{attribute addProperty BoxType "EL6861-0000-0016"}
{attribute addProperty Id "Transmit_requestBIT10.1251Receive_acceptedBIT10.1252Init_requestBIT10.1253Send_continuousBIT10.1254Output_lenUSINT819"}
{attribute addProperty CRC "829288253"}
{attribute addProperty SizeInBites "16"}
{attribute addProperty SizeInBytes "2"}
TYPE Ctrl_316DEF3D :
STRUCT
	{attribute addProperty Name "Transmit_request"}
	Transmit_request : BIT;
	{attribute addProperty Name "Receive_accepted"}
	Receive_accepted : BIT;
	{attribute addProperty Name "Init_request"}
	Init_request : BIT;
	{attribute addProperty Name "Send_continuous"}
	Send_continuous : BIT;
	{attribute 'hide'}
	reserve_1_BIT_0 : BIT;
	{attribute 'hide'}
	reserve_1_BIT_1 : BIT;
	{attribute 'hide'}
	reserve_1_BIT_2 : BIT;
	{attribute 'hide'}
	reserve_1_BIT_3 : BIT;
	{attribute addProperty Name "Output_len"}
	Output_len : USINT;
END_STRUCT
END_TYPE

(* stored: Version 1.2.0.0, ProductVersion 3.1.4024.9
   DUT Ctrl_316DEF3D: Id {deaa3ed4-9f15-491d-a575-4c4d84821476} *)
